(* Logix 5000 project; controller Savage_Saw vendor 1 type 14 code 152 rev 37.11; software revision 37.01 *)

TASK MainTask (continuous, watchdog 500 ms) : MainProgram, Inputs

MODULES
   Local : vendor 1 type 14 code 152 (PointIO 0, rev 37.11)
      Kane : vendor 590 type 43 code 5 (Ethernet 192.168.3.12, rev 1.1, StandardDataDriven RPI 20 ms)
      RemoteHPU : 1734-AENTR (Ethernet 192.168.3.11, rev 7.13, Output RPI 20 ms)
         AnalogIn5_6 : 1734-IE2V (PointIO 1, rev 3.5, Input RPI 80 ms)
         InputDC0_8 : 1734-IB8 (PointIO 3, rev 3.22)
          : 1734-IB8 (PointIO 2, rev 3.1)
          : 1734-IB8 (PointIO 4, rev 3.1)
         OutputDC0_3 : vendor 1 type 7 code 134 (PointIO 5, rev 3.2)
         OutputDC4_7 : vendor 1 type 7 code 134 (PointIO 6, rev 3.2)
      Analog0_1 : 1734-IE2V (PointIO 2, rev 3.5, Input RPI 80 ms)
      Analog2_3 : 1734-IE2V (PointIO 3, rev 3.4, Input RPI 80 ms)
      Analog4_5 : 1734-IE2V (PointIO 4, rev 3.1, Input RPI 80 ms)
      Discrete_IO : Embedded (PointIO 1, rev 37.11, Output RPI 20 ms)
      SpindleControl : 1734-OE2V (PointIO 5, rev 3.1, Output RPI 80 ms)
       : 1734-OA4 (PointIO 6, rev 3.22, Output RPI 20 ms)
       : 1734-OA4 (PointIO 7, rev 3.1, Output RPI 20 ms)
       : 1734-OA4 (PointIO 8, rev 3.1, Output RPI 20 ms)
END_MODULES

TYPE Kane_OUT_DATA1 :
STRUCT
   Unassigned_Var_Table_12 : REAL;
   Unassigned_Var_Table_13 : REAL;
   Unassigned_Var_Table_14 : REAL;
   Unassigned_Var_Table_15 : REAL;
   Unassigned_Var_Table_16 : REAL;
   Unassigned_Var_Table_17 : REAL;
   Unassigned_Var_Table_18 : REAL;
   Unassigned_Var_Table_19 : REAL;
   Unassigned_Var_Table_20 : REAL;
   Unassigned_Var_Table_21 : REAL;
END_STRUCT
END_TYPE

TYPE RMC_IN :
STRUCT
   xCutStatus : DINT;
   yBedStatus : DINT;
   zDepthStatus : DINT;
   xCutPosition : REAL;
   yBedPosition : REAL;
   zDepthPosition : REAL;
END_STRUCT
END_TYPE

TYPE RMC_OUT :
STRUCT
   xCutPosnCommand : REAL;
   yBedPosnCommand : REAL;
   zDepthPosnCommand : REAL;
   xCutVelocity : REAL;
   yBedVelocity : REAL;
   zDepthVelocity : REAL;
END_STRUCT
END_TYPE

VAR_GLOBAL   (* controller tags *)
   InBackGaugePot : ALIAS FOR Local:3:I.Ch1Data;
   inMS1HydraulicPump : ALIAS FOR Local:1:I.Data.1;
   inMS2HydraulicLoopPump : ALIAS FOR Local:1:I.Data.2;
   InMS3HydCoolingFan : ALIAS FOR Local:1:I.Data.3;
   inMS4CoolantPump : ALIAS FOR Local:1:I.Data.4;
   inMS5SwarfPump : ALIAS FOR Local:1:I.Data.5;
   inMS6SwarfConveyor : ALIAS FOR Local:1:I.Data.6;
   inRaiseLowerPot : ALIAS FOR Local:2:I.Ch1Data;
   inSpindleAside : ALIAS FOR Local:4:I.Ch0Data;
   inSpindleBside : ALIAS FOR Local:4:I.Ch1Data;
   inSpindleSpeed : ALIAS FOR Local:2:I.Ch0Data;
   inSR1SafetyRelay : ALIAS FOR Local:1:I.Data.0;
   inTraversePot : ALIAS FOR Local:3:I.Ch0Data;
   outLaserLine : ALIAS FOR Local:8:O.Data.0;
   outMS1HydraulicPump : ALIAS FOR Local:6:O.Data.0;
   outMS2HydraulicLoopPump : ALIAS FOR Local:6:O.Data.1;
   outMS3HydraulicCoolingFan : ALIAS FOR Local:6:O.Data.2;
   outMS4CoolantPump : ALIAS FOR Local:6:O.Data.3;
   outMS5SwarfPump : ALIAS FOR Local:7:O.Data.0;
   outMS6SwarfConveyor : ALIAS FOR Local:7:O.Data.1;
   outSpindleMotor : ALIAS FOR Local:5:O.Ch1Data;
   outSpindlePump : ALIAS FOR Local:5:O.Ch0Data;
   outStackLtAmber : ALIAS FOR Local:8:O.Data.2;
   outStackLtGreen : ALIAS FOR Local:8:O.Data.1;
   outStackLtRed : ALIAS FOR Local:8:O.Data.3;
   RMC_Busy : BOOL;
   RMC_In : RMC_IN := (xCutStatus := 67113540, yBedStatus := 67113540, zDepthStatus := 1108831372, xCutPosition := 37.856003);
   RMC_Out : RMC_OUT := (xCutPosnCommand := 9.999, yBedPosnCommand := 2.2, zDepthPosnCommand := 3.3, xCutVelocity := 4.4, yBedVelocity := 5.5, zDepthVelocity := 69.6);
   RMC_SendRequest : BOOL;
   tbA1JogIn : BOOL;
   tbA1JogOut : BOOL;
   tbA2JogMinus : BOOL;
   tbA3JogMinus : BOOL;
   tbA3JogPlus : BOOL;
   tbAutoCut : BOOL;
   tbAutoGage : BOOL;
   tbAutoWet : BOOL;
   tbBladeChange : BOOL;
   tbBladeCompensation : BOOL;
   tbBladeMeasure : BOOL;
   tbCCW : BOOL;
   tbCoolant : BOOL;
   tbCW : BOOL;
   tbDryBump : BOOL;
   tbDryDist : BOOL;
   tbLaser : BOOL;
   tbMS1HydPump : BOOL;
   tbMS2LoopPump : BOOL;
   tbMS3HydCoolingFan : BOOL;
   tbMS4CoolantPump : BOOL;
   tbMS5SwarfPump : BOOL;
   tbMS6SwarfConveyor : BOOL;
   tbNorthRef : BOOL;
   tbOnOff : BOOL;
   tbPlateMeasure : BOOL;
   tbSouthRef : BOOL;
   tbWetBump : BOOL;
   tbWetDistance : BOOL;
   test : DINT;
   tmrTest : TIMER := (PRE := 1000);
   X_AutoCut : BOOL;
   X_AutoGauge : BOOL;
   X_BladeChange : BOOL;
   X_BladeMeasure : BOOL;
   X_Fault : BOOL;
   X_Homing : BOOL;
   X_Manual : BOOL;
   X_Off : BOOL;
END_VAR

PROGRAM Inputs   (* main routine Main *)

ROUTINE inAnalog   (* ladder *)
END_ROUTINE

ROUTINE Main   (* ladder *)
END_ROUTINE
END_PROGRAM

PROGRAM MainProgram   (* main routine Main *)

ROUTINE Main   (* ladder *)
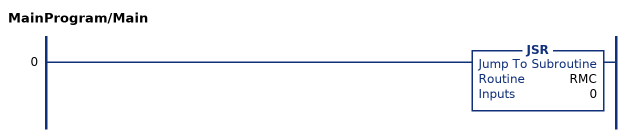
   0: JSR(RMC,0);
END_ROUTINE

ROUTINE RMC   (* ladder *)
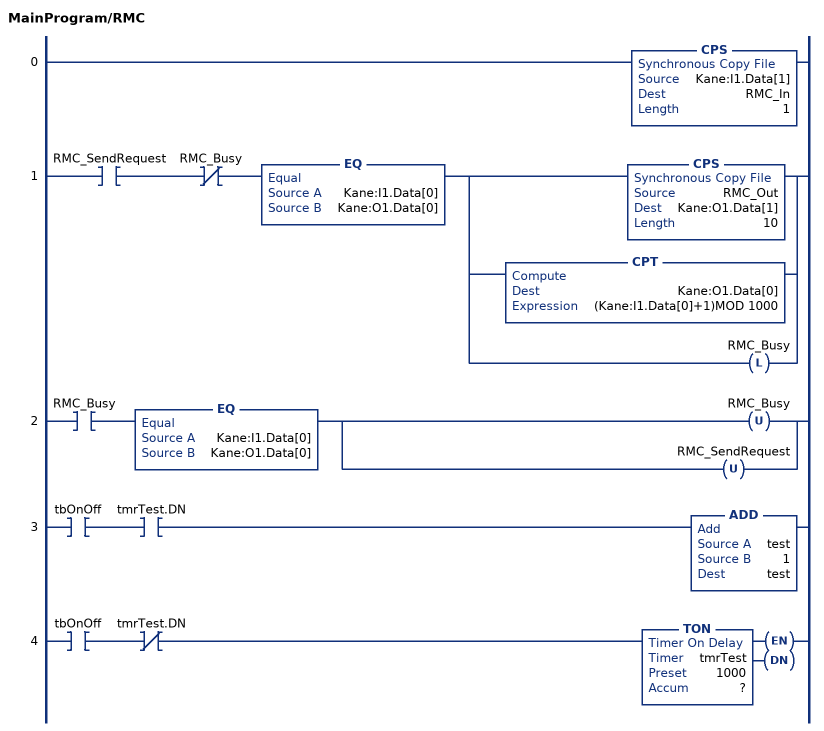
   0: CPS(Kane:I1.Data[1],RMC_In,1);
   1: XIC(RMC_SendRequest)XIO(RMC_Busy)EQ(Kane:I1.Data[0],Kane:O1.Data[0])[CPS(RMC_Out,Kane:O1.Data[1],10) ,CPT(Kane:O1.Data[0],(Kane:I1.Data[0]+1)MOD 1000) ,OTL(RMC_Busy) ];
   2: XIC(RMC_Busy)EQ(Kane:I1.Data[0],Kane:O1.Data[0])[OTU(RMC_Busy) ,OTU(RMC_SendRequest) ];
   3: XIC(tbOnOff)XIC(tmrTest.DN)ADD(test,1,test);
   4: XIC(tbOnOff)XIO(tmrTest.DN)TON(tmrTest,?,?);
END_ROUTINE
END_PROGRAM
